TYPE CTH_LA02 :
STRUCT
	Settings: GreenMasterSettingsCTH2; // Settings for the GreenMaster unit
	Status: GreenMasterStatusCTH2; // Status for the GreenMaster unit
END_STRUCT
END_TYPE

(* stored: Version 1.1.0.1, ProductVersion 3.1.4024.6
   DUT CTH_LA02: Id {efbe37fb-7a1e-494b-b09d-bcad88bf640e} *)
